PROGRAM MAIN
VAR
	bTest				: BOOL;
END_VAR

;

END_PROGRAM

(* stored: Version 1.1.0.1, ProductVersion 3.1.4026.11
   POU MAIN: Id {87d89bef-710a-4675-87ea-8ba2eeb85e21}, SpecialFunc None *)
